   MachineConfig[14]."Unit Dch"."EM - 222"."TT222-1".CW.ENABLE := True;
   MachineConfig[14]."Unit Dch"."EM - 222"."TT222-1".Address := 182;
   MachineConfig[14]."Unit Dch"."EM - 300"."AV301-1".FB_OPN_ADD := 213;
   MachineConfig[14]."Unit Dch"."EM - 300"."AV301-1".FB_CLS_ADD := 212;
   MachineConfig[14]."Unit Dch"."EM - 300"."AV301-1".ACT_OUT_ADD := 185;
   MachineConfig[14]."Unit Dch"."EM - 300"."AV302-1".TAG := 'AV635b-1';
   MachineConfig[14]."Unit Dch"."EM - 300"."AV302-1".CW.ENABLE := True;
   MachineConfig[14]."Unit Dch"."EM - 300"."AV302-1".ACT_OUT_ADD := 330;
   MachineConfig[14]."Unit Dch"."EM - 300"."AV303-1".CW.ENABLE := True;
   MachineConfig[14]."Unit Dch"."EM - 300"."AV303-1".ACT_OUT_ADD := 320;
   MachineConfig[14]."Unit Dch"."EM - 300"."AV304-1".CW.ENABLE := True;
   MachineConfig[14]."Unit Dch"."EM - 300"."AV304-1".ACT_OUT_ADD := 321;
   MachineConfig[14]."Unit Dch"."EM - 300"."AV305-1".CW.ENABLE := True;
   MachineConfig[14]."Unit Dch"."EM - 300"."AV305-1".ACT_OUT_ADD := 322;
   MachineConfig[14]."Unit Dch"."EM - 300"."AV306-1".CW.ENABLE := True;
   MachineConfig[14]."Unit Dch"."EM - 300"."AV306-1".ACT_OUT_ADD := 323;
   MachineConfig[14]."Unit Dch"."EM - 300"."AV320-1".CW.ENABLE := True;
   MachineConfig[14]."Unit Dch"."EM - 300"."AV320-1".FB_OPN_ADD := 215;
   MachineConfig[14]."Unit Dch"."EM - 300"."AV320-1".FB_CLS_ADD := 214;
   MachineConfig[14]."Unit Dch"."EM - 300"."AV320-1".ACT_OUT_ADD := 186;
   MachineConfig[14]."Unit Dch"."EM - 300"."AV635-1".TAG := 'AV635a-1';
   MachineConfig[14]."Unit Dch"."EM - 300"."AV635-1".CW.ENABLE := True;
   MachineConfig[14]."Unit Dch"."EM - 300"."AV635-1".ACT_OUT_ADD := 327;
   MachineConfig[14]."Unit Dch"."EM - 375"."AV37X-1".ACT_OUT_ADD := 324;
   MachineConfig[14]."Unit Dch"."EM - 375"."PT37X-1".CW.ENABLE := True;
   MachineConfig[14]."Unit Dch"."EM - 375"."PT37X-1".Address := 80;
   MachineConfig[14]."Unit Dch"."EM - 506"."AV543-1".CW.ENABLE := True;
   MachineConfig[14]."Unit Dch"."EM - 506"."AV543-1".FB_OPN_ADD := 230;
   MachineConfig[14]."Unit Dch"."EM - 506"."AV543-1".FB_CLS_ADD := 231;
   MachineConfig[14]."Unit Dch"."EM - 506"."AV543-1".ACT_OUT_ADD := 194;
   MachineConfig[14]."Unit Dch"."EM - 506".IP506a.CW.ENABLE := True;
   MachineConfig[14]."Unit Dch"."EM - 506"."PV376-1".CW.ENABLE := True;
   MachineConfig[14]."Unit Dch"."EM - 506"."PV376-1".ACT_OUT_ADD := 337;
   MachineConfig[14]."Unit Dch"."EM - 506"."PV376-2".CW.ENABLE := True;
   MachineConfig[14]."Unit Dch"."EM - 506"."PV376-2".CW.NO := True;
   MachineConfig[14]."Unit Dch"."EM - 506"."PV376-2".ACT_OUT_ADD := 340;
   MachineConfig[14]."Unit Dch"."EM - 506".AVDCH.ACT_OUT_ADD := 332;
   MachineConfig[14].Options."EM - 208"."AV208-1".FB_OPN_ADD := 195;
   MachineConfig[14].Options."EM - 208"."AV208-1".FB_CLS_ADD := 194;
   MachineConfig[14].Options."EM - 208"."AV208-1".ACT_OUT_ADD := 176;
   MachineConfig[14].Options."EM - 208"."FIT208-1"."Type" := 2;
   MachineConfig[14].Options."EM - 208"."FIT208-1".Address := 266;
   MachineConfig[14].Options."EM - 208"."FIT208-1".Max := 20000.0;
   MachineConfig[14].Options."EM - 210"."AV210-1".FB_OPN_ADD := 197;
   MachineConfig[14].Options."EM - 210"."AV210-1".FB_CLS_ADD := 196;
   MachineConfig[14].Options."EM - 210"."AV210-1".ACT_OUT_ADD := 177;
   MachineConfig[14].Options."EM - 463"."AV305-2".ACT_OUT_ADD := 345;
   MachineConfig[14].Options."EM - 463"."AV463-1".FB_OPN_ADD := 232;
   MachineConfig[14].Options."EM - 463"."AV463-1".FB_CLS_ADD := 233;
   MachineConfig[14].Options."EM - 463"."AV463-1".ACT_OUT_ADD := 195;
   MachineConfig[14].Options."EM - 463"."AV463-2".FB_OPN_ADD := 235;
   MachineConfig[14].Options."EM - 463"."AV463-2".FB_CLS_ADD := 234;
   MachineConfig[14].Options."EM - 463"."AV463-2".ACT_OUT_ADD := 196;
   MachineConfig[14].Options."EM - 463"."AV470-1".CW.NO := True;
   MachineConfig[14].Options."EM - 463"."AV470-1".ACT_OUT_ADD := 342;
   MachineConfig[14].Options."EM - 463"."AV660-1".ACT_OUT_ADD := 341;
   MachineConfig[14].Options."EM - 463"."AV660-2".ACT_OUT_ADD := 346;
   MachineConfig[14].Options."EM - 463"."PIT463-1".Max := 152.0;
   MachineConfig[14].Communications."EM - BC-COMM".BCI0 := 8;
   MachineConfig[14].Communications."EM - BC-COMM".BCI1 := 8;
   MachineConfig[14].Communications."EM - BC-COMM".BCI2 := 8;
   MachineConfig[14].Communications."EM - BC-COMM".BCI3 := 8;
   MachineConfig[14].Communications."EM - BC-COMM".BCO0 := 8;
   MachineConfig[14].Communications."EM - BC-COMM".BCO1 := 8;
   MachineConfig[14].Communications."EM - BC-COMM".BCO2 := 8;
   MachineConfig[14].Communications."EM - BC-COMM".BCO3 := 8;
   MachineConfig[14].Communications."EM - BC-COMM".ALARM := 8;
   MachineConfig[15].Communications."EM - BC-COMM".BCI0 := 8;
   MachineConfig[15].Communications."EM - BC-COMM".BCI1 := 8;
   MachineConfig[15].Communications."EM - BC-COMM".BCI2 := 8;
   MachineConfig[15].Communications."EM - BC-COMM".BCI3 := 8;
   MachineConfig[15].Communications."EM - BC-COMM".BCO0 := 8;
   MachineConfig[15].Communications."EM - BC-COMM".BCO1 := 8;
   MachineConfig[15].Communications."EM - BC-COMM".BCO2 := 8;
   MachineConfig[15].Communications."EM - BC-COMM".BCO3 := 8;
   MachineConfig[15].Communications."EM - BC-COMM".ALARM := 8;

END_DATA_BLOCK

